Universal Robots PolyScope program: pos6.urp

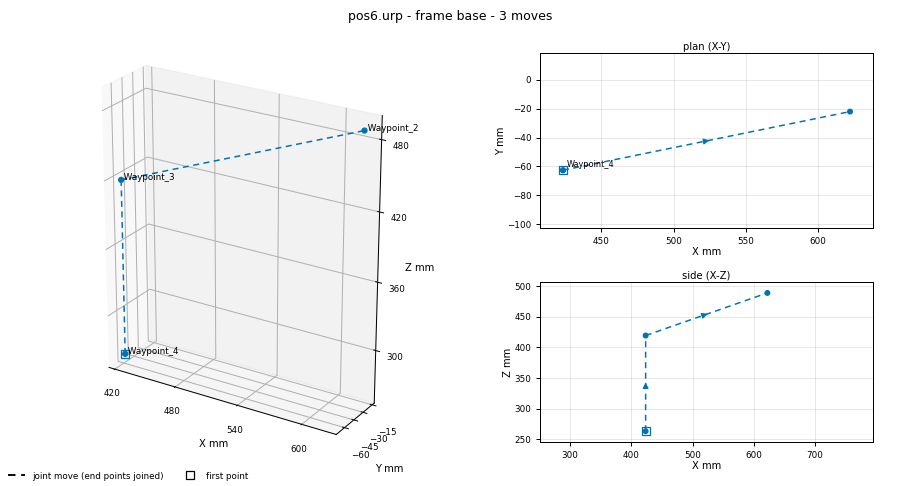
[picture p0: tool path of pos6.urp in frame base, 3 of 3 moves have a stored position in this frame; points joined in program order, loops and branches not executed]
Program pos6 (installation=default directory=/programs/Nicolas_Arteaga/quality createdIn=5.12.4.1101661 lastSavedIn=5.12.4.1101661 robotSerialNumber=20225502378)
Calibrated DH parameters: a=[0.00022, -0.425328, -0.389701, 0.000059, 0.000065, 0]; d=[0.162608, 0.803456, 9.992211, -10.662202, 0.099702, 0.099559]; alpha=[1.570756, 0.001543, 0.004316, 1.570651, -1.570122, 0]; deltaTheta=[0, 0.002917, 0.116094, -0.119008, 0, -0.000001]
Robot Program (runOnlyOnce=true)
  MoveJ speed 60 deg/s, acceleration 80 deg/s^2 (useActiveTCP=true) feature=Base
    Waypoint Waypoint_4: TCP in base x=423.413 y=-62.623 z=263.322 mm, rx=-2.7082 ry=-1.5112 rz=-0.0977 rad; joints [150.412, -75.414, 78.346, 87.06, 85.5, 2.038] deg; TCP offset x=0 y=0 z=191.5 mm, rx=0 ry=0 rz=0 rad
    Waypoint Waypoint_3: TCP in base x=423.433 y=-62.575 z=419.467 mm, rx=-2.7081 ry=-1.5114 rz=-0.0978 rad; joints [150.374, -71.697, 50.193, 111.504, 85.496, 1.888] deg
    Waypoint Waypoint_2: TCP in base x=622.09 y=-21.999 z=488.949 mm, rx=0.729 ry=1.5781 rz=1.7949 rad; joints [135.515, -94.567, 106.176, -67.801, 9.2, 55.784] deg
    'Finish Pressure Measurements'
